// Represents the milliseconds of the current second, ranging from 0 to 999.
TYPE T_Millisecond : UINT(0..999); END_TYPE

(* stored: Version 1.1.0.1
   DUT T_Millisecond: Id {7b27189b-b860-083b-04ae-fc74ce455fbf} *)
